// TIA Portal V19 export
VAR_GLOBAL   // PLC tag table "LocalMP"
   PB_Green_1500 AT %I0.0 : Bool;
   PB_Blue_1500 AT %I0.1 : Bool;
   POT1_Upper_1500 AT %IW6 : Int;   // connected to AI channel 2
   POT2_Lower_1500 AT %IW14 : Int;   // connected to AI channel 6
END_VAR
